// TIA Portal V19 export
DATA_BLOCK "ControlNodes"   // DB67
// stored: Access Published, MemoryReserve 100, Namespace Unit2.EM2
   VAR
      em { ExternalWritable := 'False'} : "LAF_typeEmControlNode";
      jobs { ExternalWritable := 'False'} : "LAF_typeJobs";
      sequence { ExternalWritable := 'False'} : "LAF_typeSequence";
      cm1Vfd206 : "LEXCHANGETRAY_typeRollerVfdContronNode";
      cm2TrayLiftingCylinder { S7_SetPoint := 'True'} : "LBC_Simple_typeTwoWayActuatorControlNode";
      cm3CellLiftingCylinder { S7_SetPoint := 'True'} : "LBC_Simple_typeTwoWayActuatorControlNode";
      cm4PositioningPinCylinder { S7_SetPoint := 'True'} : "LBC_Simple_typeTwoWayActuatorControlNode";
      cm5AxisControl : "LBC_typeAxisSimpleControlNode_1";
      cm6SignalTM { S7_SetPoint := 'True'} : "LEXCHANGETRAY_typeConstraintRollerIoSignalControlNode";
      cm7Pc { S7_SetPoint := 'True'} : "LEXCHANGETRAY_typePc_controlNode";
      cm8Scanner { S7_SetPoint := 'True'} : "LEXCHANGETRAY_typeSR1000ControlNode";
      stepCondition { S7_SetPoint := 'True'} : "LEXCHANGETRAY_typeConstraintRollerTranserfCondition";
   END_VAR
BEGIN
   em.status.enabled := true;
END_DATA_BLOCK
